FUNCTION_BLOCK FB_HMISimulationJoystick
VAR_INPUT	
END_VAR
VAR_OUTPUT
END_VAR
VAR
END_VAR



// Signal to valve
HMIoutput.fHMIControlValveSignal := HMIinput.fHMIJoystick;

END_FUNCTION_BLOCK

(* stored: Version 1.1.0.1, ProductVersion 3.1.4024.10
   POU FB_HMISimulationJoystick: Id {97020c3b-198f-42af-964f-b4237493cb4a}, SpecialFunc None *)
